FUNCTION_BLOCK OrderedDicKeyValueForwardEnumerator_TestSuite EXTENDS TcUnit.FB_TestSuite
VAR
END_VAR

CheckIsValidAtStart();
CheckKey();
CheckMoveNextReturnsFalseAtTheEnd();
CheckMoveNextReturnsTrueSingleItem();
CheckMoveNextReturnsFalseWhenEmpty();
CheckMoveNextReturnsTrueMultipleItems();
CheckReset();
CheckTryGet();
CheckTryGetTo();
CheckWorksWithArrays();
CheckWorksWithIntegers();
CheckWorksWithStrings();

METHOD PRIVATE CheckIsValidAtStart
VAR
	result : BOOL;
	dictionary : OrderedDictionary;
	enumerator : I_KeyValueForwardEnumerator;
END_VAR
TEST('CheckIsValidAtStart');

enumerator := dictionary.GetKeyValueEnumerator();

result := enumerator.IsValid;
enumerator.Dispose();

AssertTrue(
	Condition := result,
	Message := 'IsValid returned false'
);

TEST_FINISHED();
END_METHOD

METHOD PRIVATE CheckKey
VAR
	in1 : STRING := 'test1';
	in2 : STRING := 'test2';
	in3 : STRING := 'test3';
	out1 : STRING;
	out2 : STRING;
	out3 : STRING;
	expected1 : STRING := 'a';
	expected2 : STRING := 'b';
	expected3 : STRING := 'c';
	dictionary : OrderedDictionary;
	enumerator : I_KeyValueForwardEnumerator;
END_VAR
TEST('CheckKey');

dictionary.TryAdd('a',in1);
dictionary.TryAdd('b',in2);
dictionary.TryAdd('c',in3);

enumerator := dictionary.GetKeyValueEnumerator();

enumerator.MoveNext();
out1 := enumerator.Key;
enumerator.MoveNext();
out2 := enumerator.Key;
enumerator.MoveNext();
out3 := enumerator.Key;

enumerator.Dispose();

AssertEquals(
	Expected := expected1,
	Actual := out1,
	Message := 'Did not produce the expected 1st key'
);

AssertEquals(
	Expected := expected2,
	Actual := out2,
	Message := 'Did not produce the expected 2nd key'
);

AssertEquals(
	Expected := expected3,
	Actual := out3,
	Message := 'Did not produce the expected 3rd key'
);

TEST_FINISHED();
END_METHOD

METHOD PRIVATE CheckMoveNextReturnsFalseAtTheEnd
VAR
	in1 : INT := 123;
	result : BOOL;
	dictionary : OrderedDictionary;
	enumerator : I_KeyValueForwardEnumerator;
END_VAR
TEST('CheckMoveNextReturnsFalseAtTheEnd');

dictionary.TryAdd('a',in1);
enumerator := dictionary.GetKeyValueEnumerator();

enumerator.MoveNext();
result := enumerator.MoveNext();

enumerator.Dispose();

AssertFalse(result,
    'MoveNext did not correctly signal the end of the enumeration');
	
TEST_FINISHED();
END_METHOD

METHOD PRIVATE CheckMoveNextReturnsFalseWhenEmpty
VAR
	result : BOOL;
	dictionary : OrderedDictionary;
	enumerator : I_KeyValueForwardEnumerator;
	count : DINT;
END_VAR
TEST('CheckMoveNextReturnsFalseWhenEmpty');

count := dictionary.Count;
enumerator := dictionary.GetKeyValueEnumerator();

result := enumerator.MoveNext();
enumerator.Dispose();

AssertFalse(Condition := result,
    Message := 'MoveNext did not correctly signal the end of the enumeration');

TEST_FINISHED();
END_METHOD

METHOD PRIVATE CheckMoveNextReturnsTrueMultipleItems
VAR
	in1 : INT := 123;
	in2 : INT := 456;
	in3 : INT := 789;
	result : BOOL;
	dictionary : OrderedDictionary;
	enumerator : I_KeyValueForwardEnumerator;
END_VAR
TEST('CheckMoveNextReturnsTrueMultipleItems');

dictionary.TryAdd('a',in1);
dictionary.TryAdd('b',in2);
dictionary.TryAdd('c',in3);
enumerator := dictionary.GetKeyValueEnumerator();

result := enumerator.MoveNext();
enumerator.Dispose();

AssertTrue(result, 'MoveNext did not correctly signal there were more items to follow');

TEST_FINISHED();
END_METHOD

METHOD PRIVATE CheckMoveNextReturnsTrueSingleItem
VAR
	in1 : INT := 123;
	result : BOOL;
	dictionary : OrderedDictionary;
	enumerator : I_KeyValueForwardEnumerator;
END_VAR
TEST('CheckMoveNextReturnsTrueSingleItem');

dictionary.TryAdd('a',in1);
enumerator := dictionary.GetKeyValueEnumerator();

result := enumerator.MoveNext();
enumerator.Dispose();

AssertTrue(result,
    'MoveNext did not correctly signal there were more items to follow');
	
TEST_FINISHED();
END_METHOD

METHOD PRIVATE CheckReset
VAR
	in1 : ARRAY [0..1] OF REAL := [0.1,2.3];
	in2 : ARRAY [0..1] OF REAL := [1.2,3.4];
	in3 : ARRAY [0..1] OF REAL := [2.3,4.5];
	out : ARRAY [0..1] OF REAL;
	expected : ARRAY [0..1] OF REAL := [0.1,2.3];
	dictionary : OrderedDictionary;
	enumerator : I_KeyValueForwardEnumerator;
END_VAR
TEST('CheckReset');

dictionary.TryAdd('a',in1);
dictionary.TryAdd('b',in2);
dictionary.TryAdd('c',in3);

enumerator := dictionary.GetKeyValueEnumerator();

enumerator.MoveNext();
enumerator.MoveNext();
enumerator.Reset();
enumerator.MoveNext();
enumerator.TryGet(out);

enumerator.Dispose();

AssertEquals(
	Expected := expected,
	Actual := out,
	Message := 'Did not produce the expected result'
);

TEST_FINISHED();
END_METHOD

METHOD PRIVATE CheckTryGet
VAR
	in : INT := 123;
	out : INT;
	expected : INT := 123;
	result : BOOL;
	dictionary : OrderedDictionary;
	enumerator : I_KeyValueForwardEnumerator;
END_VAR
TEST('CheckTryGet');

dictionary.TryAdd('a',in);
enumerator := dictionary.GetKeyValueEnumerator();
enumerator.MoveNext();

result := enumerator.TryGet(out);
enumerator.Dispose();

AssertTrue(
	Condition := result,
	Message := 'Method returned false'
);

AssertEquals(
	Expected := expected,
	Actual := out,
	Message := 'Did not produce the expected result'
);

TEST_FINISHED();
END_METHOD

METHOD PRIVATE CheckTryGetTo
VAR
	in : INT := 123;
	out : INT;
	expected : INT := 123;
	result : BOOL;
	dictionary : OrderedDictionary;
	enumerator : I_KeyValueForwardEnumerator;
END_VAR
TEST('CheckTryGetTo');

dictionary.TryAdd('a',in);
enumerator := dictionary.GetKeyValueEnumerator();
enumerator.MoveNext();

result := enumerator.TryGetTo(ADR(out),SIZEOF(out));
enumerator.Dispose();

AssertTrue(
	Condition := result,
	Message := 'Method returned false'
);

AssertEquals(
	Expected := expected,
	Actual := out,
	Message := 'Did not produce the expected result'
);

TEST_FINISHED();
END_METHOD

METHOD PRIVATE CheckWorksWithArrays
VAR
	in1 : ARRAY [0..1] OF REAL := [0.1,2.3];
	in2 : ARRAY [0..1] OF REAL := [1.2,3.4];
	in3 : ARRAY [0..1] OF REAL := [2.3,4.5];
	out1 : ARRAY [0..1] OF REAL;
	out2 : ARRAY [0..1] OF REAL;
	out3 : ARRAY [0..1] OF REAL;
	expected1 : ARRAY [0..1] OF REAL := [0.1,2.3];
	expected2 : ARRAY [0..1] OF REAL := [1.2,3.4];
	expected3 : ARRAY [0..1] OF REAL := [2.3,4.5];
	dictionary : OrderedDictionary;
	enumerator : I_KeyValueForwardEnumerator;
END_VAR
TEST('CheckWorksWithArrays');

dictionary.TryAdd('c',in1);
dictionary.TryAdd('b',in2);
dictionary.TryAdd('a',in3);

enumerator := dictionary.GetKeyValueEnumerator();

enumerator.MoveNext();
enumerator.TryGet(out1);
enumerator.MoveNext();
enumerator.TryGet(out2);
enumerator.MoveNext();
enumerator.TryGet(out3);

enumerator.Dispose();

AssertEquals(
	Expected := expected1,
	Actual := out1,
	Message := 'Did not produce the expected 1st result'
);

AssertEquals(
	Expected := expected2,
	Actual := out2,
	Message := 'Did not produce the expected 2nd result'
);

AssertEquals(
	Expected := expected3,
	Actual := out3,
	Message := 'Did not produce the expected 3rd result'
);

TEST_FINISHED();
END_METHOD

METHOD PRIVATE CheckWorksWithIntegers
VAR
	in1 : INT := 123;
	in2 : INT := 234;
	in3 : INT := 345;
	out1 : INT;
	out2 : INT;
	out3 : INT;
	expected1 : INT := 123;
	expected2 : INT := 234;
	expected3 : INT := 345;
	dictionary : OrderedDictionary;
	enumerator : I_KeyValueForwardEnumerator;
END_VAR
TEST('CheckWorksWithIntegers');

dictionary.TryAdd('c',in1);
dictionary.TryAdd('b',in2);
dictionary.TryAdd('a',in3);

enumerator := dictionary.GetKeyValueEnumerator();

enumerator.MoveNext();
enumerator.TryGet(out1);
enumerator.MoveNext();
enumerator.TryGet(out2);
enumerator.MoveNext();
enumerator.TryGet(out3);

enumerator.Dispose();

AssertEquals(
	Expected := expected1,
	Actual := out1,
	Message := 'Did not produce the expected 1st result'
);

AssertEquals(
	Expected := expected2,
	Actual := out2,
	Message := 'Did not produce the expected 2nd result'
);

AssertEquals(
	Expected := expected3,
	Actual := out3,
	Message := 'Did not produce the expected 3rd result'
);

TEST_FINISHED();
END_METHOD

METHOD PRIVATE CheckWorksWithStrings
VAR
	in1 : STRING := 'test1';
	in2 : STRING := 'test2';
	in3 : STRING := 'test3';
	out1 : STRING;
	out2 : STRING;
	out3 : STRING;
	expected1 : STRING := 'test1';
	expected2 : STRING := 'test2';
	expected3 : STRING := 'test3';
	dictionary : OrderedDictionary;
	enumerator : I_KeyValueForwardEnumerator;
END_VAR
TEST('CheckWorksWithStrings');

dictionary.TryAdd('c',in1);
dictionary.TryAdd('b',in2);
dictionary.TryAdd('a',in3);

enumerator := dictionary.GetKeyValueEnumerator();

enumerator.MoveNext();
enumerator.TryGet(out1);
enumerator.MoveNext();
enumerator.TryGet(out2);
enumerator.MoveNext();
enumerator.TryGet(out3);

enumerator.Dispose();

AssertEquals(
	Expected := expected1,
	Actual := out1,
	Message := 'Did not produce the expected 1st result'
);

AssertEquals(
	Expected := expected2,
	Actual := out2,
	Message := 'Did not produce the expected 2nd result'
);

AssertEquals(
	Expected := expected3,
	Actual := out3,
	Message := 'Did not produce the expected 3rd result'
);

TEST_FINISHED();
END_METHOD

END_FUNCTION_BLOCK

(* stored: Version 1.1.0.1, ProductVersion 3.1.4024.12
   POU OrderedDicKeyValueForwardEnumerator_TestSuite: Id {b245bb92-7484-4d17-af3a-aa37aeccedc9}, SpecialFunc None
   Method CheckIsValidAtStart: Id {1994e45f-c17a-4cca-bf31-142fbe8345ae}
   Method CheckKey: Id {8c9b505a-1dd9-4545-b5e6-39ebcd07c832}
   Method CheckMoveNextReturnsFalseAtTheEnd: Id {8bb54452-53bc-4ce6-994c-dfd5d82e9547}
   Method CheckMoveNextReturnsFalseWhenEmpty: Id {9c6949ac-a149-431c-b3ee-3d990b998d5c}
   Method CheckMoveNextReturnsTrueMultipleItems: Id {cca16160-4900-49bf-a179-51b8fef3a800}
   Method CheckMoveNextReturnsTrueSingleItem: Id {fdb84057-9d4c-4491-a1c3-6210dd2d3ab4}
   Method CheckReset: Id {94e2fac9-6536-42c7-a7b1-fbf587dafe1f}
   Method CheckTryGet: Id {6622e031-d5c9-48a6-85fe-a40638568d2b}
   Method CheckTryGetTo: Id {28608e76-b3e3-48c5-961a-ae4c96c32674}
   Method CheckWorksWithArrays: Id {99936fdf-c08b-4cd7-9b1b-2ff7eeb4ba74}
   Method CheckWorksWithIntegers: Id {e61a0e62-2085-480e-9dd0-299cc103d6dd}
   Method CheckWorksWithStrings: Id {d77bc4f0-0a19-42c7-884a-a7ed6b16f1ed} *)
